{attribute 'call_after_init'}
FUNCTION_BLOCK FB_DumpChiller_Test EXTENDS FB_TestSuite
VAR_INPUT
END_VAR
VAR_OUTPUT
END_VAR
VAR
END_VAR

ErrorTriggers();
ErrorResets();
ErrorLatches();
NoError();

METHOD ErrorLatches
VAR
	fbDumpChiller : FB_DumpChiller := F_DumpChiller_Error();
END_VAR
TEST('ErrorLatches');

fbDumpChiller(bDumpChillerFlow := TRUE);
AssertTrue(fbDumpChiller.bError, 'Error did not latch');

TEST_FINISHED();
END_METHOD

METHOD ErrorResets
VAR
	fbDumpChiller : FB_DumpChiller := F_DumpChiller_Error();
END_VAR
TEST('ErrorResets');

fbDumpChiller.Reset();
fbDumpChiller(bDumpChillerFlow := TRUE);
AssertFalse(fbDumpChiller.bError, 'Error did not reset');

TEST_FINISHED();
END_METHOD

METHOD ErrorTriggers
VAR
	fbDumpChiller : FB_DumpChiller := F_DumpChiller_Error();
END_VAR
TEST('ErrorTriggers');

AssertTrue(fbDumpChiller.bError, 'Error did not trigger');

TEST_FINISHED();
END_METHOD

METHOD NoError
VAR
	fbDumpChiller : FB_DumpChiller;
END_VAR
TEST('NoError');

fbDumpChiller(
	bAmphosOn := TRUE,
	bDumpChillerFlow := TRUE
);
AssertFalse(fbDumpChiller.bError, 'Error falsely triggered');

TEST_FINISHED();
END_METHOD

END_FUNCTION_BLOCK

(* stored: Version 1.1.0.1, ProductVersion 3.1.4020.14
   POU FB_DumpChiller_Test: Id {53397a3d-ecaf-42b9-bc44-be2241179a62}, SpecialFunc None
   Method ErrorLatches: Id {4918d277-84e8-432c-9be5-159d999bbd74}
   Method ErrorResets: Id {4549f291-7a5a-45b8-8c94-a44d2dfa627f}
   Method ErrorTriggers: Id {8991acc0-a708-4167-8a8c-9ce91b374fbf}
   Method NoError: Id {b9104161-6218-4f80-a48b-0738e37e1166} *)
